FUNCTION_BLOCK FC_Unit (* Unit PackML state machine; only PROC may declare procedure completion; skills acknowledge hold/stop through the equipment-module status chain *)
  (* Standard: 61499-2 *)
  (* Version 2.0, 2026-09-27, Project contributors, Filling cell reference model *)
  PACKAGE fillingcell;
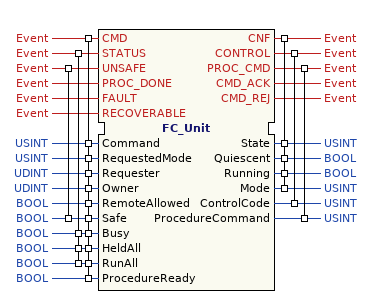
  EVENT_INPUT
    CMD WITH Command, RequestedMode, Requester, Owner, RemoteAllowed, Safe, Busy, HeldAll, RunAll, ProcedureReady;
    STATUS WITH Busy, HeldAll, RunAll;
    UNSAFE WITH Safe;
    PROC_DONE;
    FAULT;
    RECOVERABLE;
  END_EVENT
  EVENT_OUTPUT
    CNF WITH State, Quiescent, Running, Mode;
    CONTROL WITH ControlCode;
    PROC_CMD WITH ProcedureCommand;
    CMD_ACK;
    CMD_REJ;
  END_EVENT
  VAR_INPUT
    Command : USINT;
    RequestedMode : USINT;
    Requester : UDINT;
    Owner : UDINT;
    RemoteAllowed : BOOL;
    Safe : BOOL;
    Busy : BOOL;
    HeldAll : BOOL := TRUE;
    RunAll : BOOL := TRUE;
    ProcedureReady : BOOL;
  END_VAR
  VAR_OUTPUT
    State : USINT := 2;
    Quiescent : BOOL := TRUE;
    Running : BOOL;
    Mode : USINT;
    ControlCode : USINT;
    ProcedureCommand : USINT;
  END_VAR
  EC_STATES
    Stopped : Alg_Stopped -> CNF;
    Clearing : Alg_Clearing -> CNF, -> CONTROL, -> PROC_CMD;
    Starting : Alg_Starting -> CNF;
    Idle : Alg_Idle -> CNF;
    Suspended : Alg_Suspended -> CNF;
    Execute : Alg_Execute -> CNF, -> PROC_CMD;
    Stopping : Alg_Stopping -> CNF, -> CONTROL, -> PROC_CMD;
    Aborting : Alg_Aborting -> CNF, -> CONTROL, -> PROC_CMD;
    Aborted : Alg_Aborted -> CNF;
    Holding : Alg_Holding -> CNF, -> CONTROL, -> PROC_CMD;
    Held : Alg_Held -> CNF;
    Unholding : Alg_Unholding -> CNF, -> CONTROL, -> PROC_CMD;
    Suspending : Alg_Suspending -> CNF, -> CONTROL, -> PROC_CMD;
    Unsuspending : Alg_Unsuspending -> CNF, -> CONTROL, -> PROC_CMD;
    Resetting : Alg_Resetting -> CNF, -> CONTROL, -> PROC_CMD;
    Completing : Alg_Completing -> CNF;
    Complete : Alg_Complete -> CNF;
    UpdateIdle : Alg_UpdateIdle -> CNF;
    UpdateComplete : Alg_UpdateComplete -> CNF;
    UpdateStopped : Alg_UpdateStopped -> CNF;
    UpdateAborted : Alg_UpdateAborted -> CNF;
    Ack0_Resetting : -> CMD_ACK;
    Ack1_Resetting : -> CMD_ACK;
    Ack2_Resetting : -> CMD_ACK;
    Ack3_Starting : -> CMD_ACK;
    Ack4_Holding : -> CMD_ACK;
    Ack5_Unholding : -> CMD_ACK;
    Ack6_Holding : -> CMD_ACK;
    Ack7_Holding : -> CMD_ACK;
    Ack8_Holding : -> CMD_ACK;
    Ack9_Suspending : -> CMD_ACK;
    Ack10_Unsuspending : -> CMD_ACK;
    Ack11_Aborting : -> CMD_ACK;
    Ack12_Aborting : -> CMD_ACK;
    Ack13_Stopping : -> CMD_ACK;
    Ack14_Aborting : -> CMD_ACK;
    Ack15_Stopping : -> CMD_ACK;
    Ack16_Aborting : -> CMD_ACK;
    Ack17_Stopping : -> CMD_ACK;
    Ack18_Aborting : -> CMD_ACK;
    Ack19_Stopping : -> CMD_ACK;
    Ack20_Aborting : -> CMD_ACK;
    Ack21_Stopping : -> CMD_ACK;
    Ack22_Aborting : -> CMD_ACK;
    Ack23_Stopping : -> CMD_ACK;
    Ack24_Aborting : -> CMD_ACK;
    Ack25_Stopping : -> CMD_ACK;
    Ack26_Aborting : -> CMD_ACK;
    Ack27_Stopping : -> CMD_ACK;
    Ack28_Aborting : -> CMD_ACK;
    Ack29_Stopping : -> CMD_ACK;
    Ack30_Aborting : -> CMD_ACK;
    Ack31_Stopping : -> CMD_ACK;
    Ack32_Aborting : -> CMD_ACK;
    Ack33_Stopping : -> CMD_ACK;
    Ack34_Clearing : -> CMD_ACK;
    RejClearing : -> CMD_REJ;
    RejStopped : -> CMD_REJ;
    RejStarting : -> CMD_REJ;
    RejIdle : -> CMD_REJ;
    RejSuspended : -> CMD_REJ;
    RejExecute : -> CMD_REJ;
    RejStopping : -> CMD_REJ;
    RejAborting : -> CMD_REJ;
    RejAborted : -> CMD_REJ;
    RejHolding : -> CMD_REJ;
    RejHeld : -> CMD_REJ;
    RejUnholding : -> CMD_REJ;
    RejSuspending : -> CMD_REJ;
    RejUnsuspending : -> CMD_REJ;
    RejResetting : -> CMD_REJ;
    RejCompleting : -> CMD_REJ;
    RejComplete : -> CMD_REJ;
  END_STATES
  EC_TRANSITIONS
    Resetting TO Idle := STATUS[NOT Busy];
    Starting TO Execute := 1;
    Execute TO Completing := PROC_DONE;
    Completing TO Complete := 1;
    Execute TO Holding := RECOVERABLE;
    Holding TO Held := STATUS[HeldAll];
    Unholding TO Execute := STATUS[(Mode = 0) AND RunAll];
    Unholding TO Idle := STATUS[(Mode <> 0) AND RunAll];
    Suspending TO Suspended := STATUS[HeldAll];
    Unsuspending TO Execute := STATUS[RunAll];
    Stopped TO Aborting := UNSAFE;
    Idle TO Aborting := UNSAFE;
    Execute TO Aborting := UNSAFE;
    Execute TO Aborting := FAULT;
    Complete TO Aborting := UNSAFE;
    Held TO Aborting := UNSAFE;
    Held TO Aborting := FAULT;
    Suspended TO Aborting := UNSAFE;
    Suspended TO Aborting := FAULT;
    Holding TO Aborting := UNSAFE;
    Holding TO Aborting := FAULT;
    Unholding TO Aborting := UNSAFE;
    Unholding TO Aborting := FAULT;
    Suspending TO Aborting := UNSAFE;
    Suspending TO Aborting := FAULT;
    Unsuspending TO Aborting := UNSAFE;
    Unsuspending TO Aborting := FAULT;
    Resetting TO Aborting := UNSAFE;
    Stopping TO Aborting := UNSAFE;
    Stopping TO Stopped := STATUS[NOT Busy];
    Aborting TO Aborted := STATUS[NOT Busy];
    Clearing TO Stopped := STATUS[NOT Busy];
    Idle TO UpdateIdle := STATUS;
    UpdateIdle TO Idle := 1;
    Complete TO UpdateComplete := STATUS;
    UpdateComplete TO Complete := 1;
    Stopped TO UpdateStopped := STATUS;
    UpdateStopped TO Stopped := 1;
    Aborted TO UpdateAborted := STATUS;
    UpdateAborted TO Aborted := 1;
    Stopped TO Ack0_Resetting := CMD[(Command = 1) AND (RemoteAllowed AND (Requester = Owner) AND (RequestedMode <= 2)) AND NOT Busy];
    Ack0_Resetting TO Resetting := 1;
    Idle TO Ack1_Resetting := CMD[(Command = 1) AND (RemoteAllowed AND (Requester = Owner) AND (RequestedMode <= 2)) AND NOT Busy];
    Ack1_Resetting TO Resetting := 1;
    Complete TO Ack2_Resetting := CMD[(Command = 1) AND (RemoteAllowed AND (Requester = Owner) AND (RequestedMode <= 2)) AND NOT Busy];
    Ack2_Resetting TO Resetting := 1;
    Idle TO Ack3_Starting := CMD[(Command = 2) AND (RemoteAllowed AND (Requester = Owner) AND (RequestedMode <= 2)) AND Safe AND NOT Busy AND (Mode = 0) AND ProcedureReady];
    Ack3_Starting TO Starting := 1;
    Execute TO Ack4_Holding := CMD[(Command = 3) AND (RemoteAllowed AND (Requester = Owner) AND (RequestedMode <= 2))];
    Ack4_Holding TO Holding := 1;
    Held TO Ack5_Unholding := CMD[(Command = 4) AND (RemoteAllowed AND (Requester = Owner) AND (RequestedMode <= 2)) AND Safe];
    Ack5_Unholding TO Unholding := 1;
    Idle TO Ack6_Holding := CMD[(Command = 3) AND (RemoteAllowed AND (Requester = Owner) AND (RequestedMode <= 2)) AND Busy AND (Mode <> 0)];
    Ack6_Holding TO Holding := 1;
    Stopped TO Ack7_Holding := CMD[(Command = 3) AND (RemoteAllowed AND (Requester = Owner) AND (RequestedMode <= 2)) AND Busy AND (Mode <> 0)];
    Ack7_Holding TO Holding := 1;
    Complete TO Ack8_Holding := CMD[(Command = 3) AND (RemoteAllowed AND (Requester = Owner) AND (RequestedMode <= 2)) AND Busy AND (Mode <> 0)];
    Ack8_Holding TO Holding := 1;
    Execute TO Ack9_Suspending := CMD[(Command = 8) AND (RemoteAllowed AND (Requester = Owner) AND (RequestedMode <= 2))];
    Ack9_Suspending TO Suspending := 1;
    Suspended TO Ack10_Unsuspending := CMD[(Command = 9) AND (RemoteAllowed AND (Requester = Owner) AND (RequestedMode <= 2)) AND Safe];
    Ack10_Unsuspending TO Unsuspending := 1;
    Stopped TO Ack11_Aborting := CMD[Command = 6];
    Ack11_Aborting TO Aborting := 1;
    Idle TO Ack12_Aborting := CMD[Command = 6];
    Ack12_Aborting TO Aborting := 1;
    Idle TO Ack13_Stopping := CMD[Command = 5];
    Ack13_Stopping TO Stopping := 1;
    Execute TO Ack14_Aborting := CMD[Command = 6];
    Ack14_Aborting TO Aborting := 1;
    Execute TO Ack15_Stopping := CMD[Command = 5];
    Ack15_Stopping TO Stopping := 1;
    Complete TO Ack16_Aborting := CMD[Command = 6];
    Ack16_Aborting TO Aborting := 1;
    Complete TO Ack17_Stopping := CMD[Command = 5];
    Ack17_Stopping TO Stopping := 1;
    Held TO Ack18_Aborting := CMD[Command = 6];
    Ack18_Aborting TO Aborting := 1;
    Held TO Ack19_Stopping := CMD[Command = 5];
    Ack19_Stopping TO Stopping := 1;
    Suspended TO Ack20_Aborting := CMD[Command = 6];
    Ack20_Aborting TO Aborting := 1;
    Suspended TO Ack21_Stopping := CMD[Command = 5];
    Ack21_Stopping TO Stopping := 1;
    Holding TO Ack22_Aborting := CMD[Command = 6];
    Ack22_Aborting TO Aborting := 1;
    Holding TO Ack23_Stopping := CMD[Command = 5];
    Ack23_Stopping TO Stopping := 1;
    Unholding TO Ack24_Aborting := CMD[Command = 6];
    Ack24_Aborting TO Aborting := 1;
    Unholding TO Ack25_Stopping := CMD[Command = 5];
    Ack25_Stopping TO Stopping := 1;
    Suspending TO Ack26_Aborting := CMD[Command = 6];
    Ack26_Aborting TO Aborting := 1;
    Suspending TO Ack27_Stopping := CMD[Command = 5];
    Ack27_Stopping TO Stopping := 1;
    Unsuspending TO Ack28_Aborting := CMD[Command = 6];
    Ack28_Aborting TO Aborting := 1;
    Unsuspending TO Ack29_Stopping := CMD[Command = 5];
    Ack29_Stopping TO Stopping := 1;
    Resetting TO Ack30_Aborting := CMD[Command = 6];
    Ack30_Aborting TO Aborting := 1;
    Resetting TO Ack31_Stopping := CMD[Command = 5];
    Ack31_Stopping TO Stopping := 1;
    Stopping TO Ack32_Aborting := CMD[Command = 6];
    Ack32_Aborting TO Aborting := 1;
    Stopped TO Ack33_Stopping := CMD[(Command = 5) AND Busy];
    Ack33_Stopping TO Stopping := 1;
    Aborted TO Ack34_Clearing := CMD[(Command = 7) AND (RemoteAllowed AND (Requester = Owner) AND (RequestedMode <= 2)) AND Safe];
    Ack34_Clearing TO Clearing := 1;
    Clearing TO RejClearing := CMD;
    RejClearing TO Clearing := 1;
    Stopped TO RejStopped := CMD;
    RejStopped TO Stopped := 1;
    Starting TO RejStarting := CMD;
    RejStarting TO Starting := 1;
    Idle TO RejIdle := CMD;
    RejIdle TO Idle := 1;
    Suspended TO RejSuspended := CMD;
    RejSuspended TO Suspended := 1;
    Execute TO RejExecute := CMD;
    RejExecute TO Execute := 1;
    Stopping TO RejStopping := CMD;
    RejStopping TO Stopping := 1;
    Aborting TO RejAborting := CMD;
    RejAborting TO Aborting := 1;
    Aborted TO RejAborted := CMD;
    RejAborted TO Aborted := 1;
    Holding TO RejHolding := CMD;
    RejHolding TO Holding := 1;
    Held TO RejHeld := CMD;
    RejHeld TO Held := 1;
    Unholding TO RejUnholding := CMD;
    RejUnholding TO Unholding := 1;
    Suspending TO RejSuspending := CMD;
    RejSuspending TO Suspending := 1;
    Unsuspending TO RejUnsuspending := CMD;
    RejUnsuspending TO Unsuspending := 1;
    Resetting TO RejResetting := CMD;
    RejResetting TO Resetting := 1;
    Completing TO RejCompleting := CMD;
    RejCompleting TO Completing := 1;
    Complete TO RejComplete := CMD;
    RejComplete TO Complete := 1;
  END_TRANSITIONS
  ALGORITHM Alg_Stopped IN ST:
State := 2;
Running := FALSE;
Quiescent := NOT Busy;
  END_ALGORITHM
  ALGORITHM Alg_Clearing IN ST:
State := 1;
Running := FALSE;
Quiescent := FALSE;
ControlCode := 7;
ProcedureCommand := 7;
  END_ALGORITHM
  ALGORITHM Alg_Starting IN ST:
State := 3;
Running := FALSE;
Quiescent := FALSE;
ProcedureCommand := 2;
  END_ALGORITHM
  ALGORITHM Alg_Idle IN ST:
State := 4;
Running := FALSE;
Quiescent := NOT Busy;
  END_ALGORITHM
  ALGORITHM Alg_Suspended IN ST:
State := 5;
Running := FALSE;
Quiescent := FALSE;
  END_ALGORITHM
  ALGORITHM Alg_Execute IN ST:
State := 6;
Running := TRUE;
Quiescent := FALSE;
  END_ALGORITHM
  ALGORITHM Alg_Stopping IN ST:
State := 7;
Running := FALSE;
Quiescent := FALSE;
ControlCode := 5;
ProcedureCommand := 5;
  END_ALGORITHM
  ALGORITHM Alg_Aborting IN ST:
State := 8;
Running := FALSE;
Quiescent := FALSE;
ControlCode := 6;
ProcedureCommand := 6;
  END_ALGORITHM
  ALGORITHM Alg_Aborted IN ST:
State := 9;
Running := FALSE;
Quiescent := NOT Busy;
  END_ALGORITHM
  ALGORITHM Alg_Holding IN ST:
State := 10;
Running := FALSE;
Quiescent := FALSE;
ControlCode := 3;
ProcedureCommand := 3;
  END_ALGORITHM
  ALGORITHM Alg_Held IN ST:
State := 11;
Running := FALSE;
Quiescent := FALSE;
  END_ALGORITHM
  ALGORITHM Alg_Unholding IN ST:
State := 12;
Running := FALSE;
Quiescent := FALSE;
ControlCode := 4;
ProcedureCommand := 4;
  END_ALGORITHM
  ALGORITHM Alg_Suspending IN ST:
State := 13;
Running := FALSE;
Quiescent := FALSE;
ControlCode := 3;
ProcedureCommand := 8;
  END_ALGORITHM
  ALGORITHM Alg_Unsuspending IN ST:
State := 14;
Running := FALSE;
Quiescent := FALSE;
ControlCode := 4;
ProcedureCommand := 9;
  END_ALGORITHM
  ALGORITHM Alg_Resetting IN ST:
State := 15;
Running := FALSE;
Quiescent := FALSE;
Mode := RequestedMode;
ControlCode := 1;
ProcedureCommand := 1;
  END_ALGORITHM
  ALGORITHM Alg_Completing IN ST:
State := 16;
Running := FALSE;
Quiescent := FALSE;
  END_ALGORITHM
  ALGORITHM Alg_Complete IN ST:
State := 17;
Running := FALSE;
Quiescent := NOT Busy;
  END_ALGORITHM
  ALGORITHM Alg_UpdateIdle IN ST:
Quiescent := NOT Busy;
  END_ALGORITHM
  ALGORITHM Alg_UpdateComplete IN ST:
Quiescent := NOT Busy;
  END_ALGORITHM
  ALGORITHM Alg_UpdateStopped IN ST:
Quiescent := NOT Busy;
  END_ALGORITHM
  ALGORITHM Alg_UpdateAborted IN ST:
Quiescent := NOT Busy;
  END_ALGORITHM
END_FUNCTION_BLOCK
